FUNCTION_BLOCK FB_EcMasterState

VAR_INPUT
	sNetId           : T_AmsNetId; //:= '5.124.224.126.6.1';
END_VAR

VAR
    fbReqMasterState : FB_EcReqMasterState;
    bExecute         : BOOL;
	tTimeout		 : TIME := DEFAULT_ADS_TIMEOUT;
    state            : WORD;;
	bBusy  			 : BOOL;
END_VAR

VAR_OUTPUT
    bError           : BOOL;
    nErrId           : UDINT;

	bStateChangeSuccsessful : BOOL;//fertig bit
	bStateChangeOccurred : BOOL; //erfolgt bit
END_VAR

//other function blocks
VAR
	fTrig			: F_Trig;
END_VAR

fbReqMasterState(sNetId:= sNetId, bExecute:=bExecute, state:=EC_DEVICE_STATE_INIT);
bError := fbReqMasterState.bError;
nErrId := fbReqMasterState.nErrId;
bBusy := fbReqMasterState.bBusy;

fTrig(CLK := bBusy);

//wenn nicht mehr bussy dann bStateChangeOccured / succsess
IF fTrig.Q AND NOT bError THEN
	bStateChangeOccurred := TRUE;
	bStateChangeSuccsessful := TRUE;
ELSIF fTrig.Q AND NOT bError THEN
	bStateChangeOccurred := TRUE;
	bStateChangeSuccsessful := FALSE;
END_IF

{attribute 'TcRpcEnable'}
METHOD DisableMaster : BOOL
VAR_INPUT
END_VAR
IF NOT bBusy THEN
	bExecute := TRUE;
	fbReqMasterState(sNetId:= sNetId, bExecute:=bExecute, state:=EC_DEVICE_STATE_INIT);
	bExecute := FALSE;
	bError := fbReqMasterState.bError;
	nErrId := fbReqMasterState.nErrId;
	bBusy := fbReqMasterState.bBusy;
	
	bStateChangeOccurred := FALSE; //reset
	bStateChangeSuccsessful := FALSE; //reset
	
	DisableMaster := TRUE;
ELSE
	DisableMaster := FALSE;
END_IF
END_METHOD

{attribute 'TcRpcEnable'}
METHOD EnableMaster : BOOL
VAR_INPUT
END_VAR

VAR
END_VAR
IF NOT bBusy THEN
	bExecute := TRUE;
	fbReqMasterState(sNetId:= sNetId, bExecute:=bExecute, state:=EC_DEVICE_STATE_OP);
	bExecute := FALSE;
	bError := fbReqMasterState.bError;
	nErrId := fbReqMasterState.nErrId;
	bBusy := fbReqMasterState.bBusy;
	
	bStateChangeOccurred := FALSE; //reset
	bStateChangeSuccsessful := FALSE; //reset
	
	EnableMaster := TRUE;
ELSE
	EnableMaster := FALSE;
END_IF
END_METHOD

END_FUNCTION_BLOCK

(* stored: Version 1.1.0.1, ProductVersion 3.1.4024.11
   POU FB_EcMasterState: Id {405fdbf8-f334-46b0-bbce-28e2b07965a9}, SpecialFunc None
   Method DisableMaster: Id {29b01c97-b07f-4ad5-9efe-e980c6fe8cda}
   Method EnableMaster: Id {21eda505-3e42-4f35-947a-1d0981096251} *)
